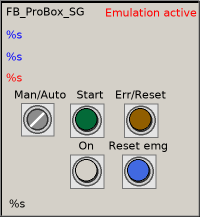
VISUALIZATION V_Group  // 200x217
VAR_IN_OUT
	{attribute 'VAR_IN_OUT_AS_POINTER'}
	fbFunction		: FB_ProBOXSG;
	fbEmuFunction	: FB_ProBOXSG_Emulation;
END_VAR
    Rectangle (0,1 200x216)
    Rectangle (6,194 177x20), "%s", text variable: fbFunction.ConfigGroup.GroupName
    Label (3,2 158x20), "FB_ProBox_SG"
    Rectangle (3,25 99x20), "%s", text variable: fbFunction.GroupData.OperationState.eState
    Rectangle (3,68 161x20), "%s", tooltip "%s", text variable: fbFunction.GroupData.ErrorData.Error.ErrorCode.Conv, invisible if: fbFunction.GroupData.ErrorData.Error.ErrorCode.Conv = 0
        p4168582468: fbFunction.GroupData.ErrorData.Error.ErrorParam
    Rectangle (3,47 99x20), "%s", text variable: fbFunction.GroupData.OperationState.eMode
    RotarySwitch (21,103 33x33), variable: fbEmuFunction.DebugManualModeSw, behaviour: TOGGLE, style: Switch-RotarySwitch-Gray
    Label (11,84 58x22), "Man/Auto"
    Rectangle (102,3 95x20), "Emulation active", invisible if: NOT ProBoxSystem.EMULATION_ENABLED
    PushSwitch (70,103 34x35), behaviour: TOGGLE, style: Switch-PushSwitch-Gray
    Ellipse (75,108 22x22), colour toggle: fbFunction.HW_Outputs.GroupStarted
        tap fbEmuFunction.DebugStartButton
    Label (71,84 38x22), "Start"
    Label (106,84 69x22), "Err/Reset"
    PushSwitch (124,103 34x35), behaviour: TOGGLE, style: Switch-PushSwitch-Gray
    Ellipse (129,108 22x22), colour toggle: fbFunction.HW_Outputs.ErrorPending
        tap fbEmuFunction.DebugResetButton
    Label (52,135 69x22), "On"
    PushSwitch (70,154 34x35), behaviour: TOGGLE, style: Switch-PushSwitch-Gray
    Ellipse (75,159 22x22), colour toggle: fbFunction.HW_Outputs.MainContactorLamp
        tap fbEmuFunction.DebugMcOnButton
    PushSwitch (122,154 34x35), behaviour: TOGGLE, style: Switch-PushSwitch-Gray
    Ellipse (127,159 22x22), colour toggle: fbFunction.HW_Outputs.EmergencyLamp
        tap fbEmuFunction.DebugResetEmgButton
    Label (104,135 69x22), "Reset emg"
END_VISUALIZATION

(* stored: Version 1.1.0.1, ProductVersion 3.1.4024.9
   Visu V_Group: Id {087c644b-ba66-4b45-88a4-70693d73f358} *)
